FUNCTION_BLOCK LuggageMove (* Basic Function Block Type *)
  (* Standard: 61499-2 *)
  (* Version 0.0, 6/23/2016, Andrei, nxtControl GmbH, Template *)
  PACKAGE Main;
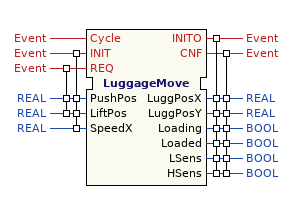
  EVENT_INPUT
    Cycle;
    INIT WITH PushPos, LiftPos, SpeedX; (* Initialization Request *)
    REQ WITH PushPos, LiftPos; (* Normal Execution Request *)
  END_EVENT
  EVENT_OUTPUT
    INITO WITH LuggPosX, LuggPosY, Loading, Loaded, LSens, HSens; (* Initialization Confirm *)
    CNF WITH LuggPosX, LuggPosY, Loading, Loaded, LSens, HSens; (* Execution Confirmation *)
  END_EVENT
  VAR_INPUT
    PushPos : REAL;
    LiftPos : REAL;
    SpeedX : REAL;
  END_VAR
  VAR_OUTPUT
    LuggPosX : REAL; (* Output event qualifier *)
    LuggPosY : REAL;
    Loading : BOOL; (* Input event qualifier *)
    Loaded : BOOL;
    LSens : BOOL;
    HSens : BOOL;
  END_VAR
  VAR
    X : REAL := 0.0;
    Y : REAL := 0.0;
    pPushPos : REAL;
    pLiftPos : REAL;
  END_VAR
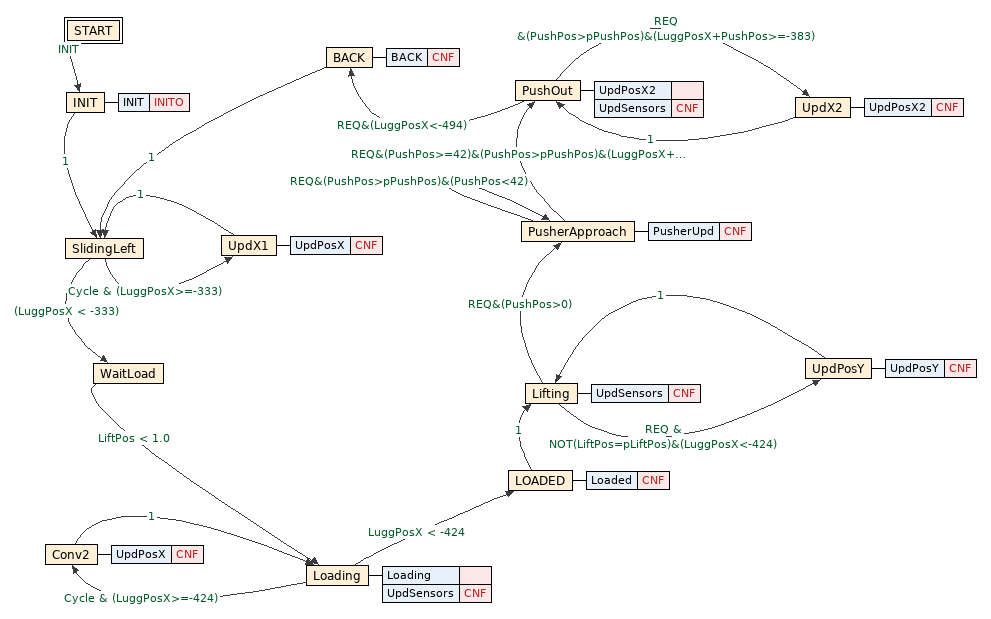
  EC_STATES
    START; (* Initial State *)
    INIT : INIT -> INITO; (* Initialization *)
    SlidingLeft; (* Normal execution *)
    UpdX1 : UpdPosX -> CNF;
    WaitLoad;
    Loading : Loading, UpdSensors -> CNF;
    Conv2 : UpdPosX -> CNF;
    Lifting : UpdSensors -> CNF;
    UpdPosY : UpdPosY -> CNF;
    PushOut : UpdPosX2, UpdSensors -> CNF;
    UpdX2 : UpdPosX2 -> CNF;
    LOADED : Loaded -> CNF;
    PusherApproach : PusherUpd -> CNF;
    BACK : BACK -> CNF;
  END_STATES
  EC_TRANSITIONS
    START TO INIT := INIT;
    INIT TO SlidingLeft := 1;
    SlidingLeft TO UpdX1 := Cycle & (LuggPosX>=-333);
    UpdX1 TO SlidingLeft := 1;
    SlidingLeft TO WaitLoad := (LuggPosX < -333);
    WaitLoad TO Loading := LiftPos < 1.0;
    Loading TO Conv2 := Cycle & (LuggPosX>=-424);
    Conv2 TO Loading := 1;
    Loading TO LOADED := LuggPosX < -424;
    UpdPosY TO Lifting := 1;
    Lifting TO UpdPosY := REQ & NOT(LiftPos=pLiftPos)&(LuggPosX<-424);
    PusherApproach TO PushOut := REQ&(PushPos>=42)&(PushPos>pPushPos)&(LuggPosX+PushPos>=-383);
    PushOut TO UpdX2 := REQ &(PushPos>pPushPos)&(LuggPosX+PushPos>=-383);
    UpdX2 TO PushOut := 1;
    LOADED TO Lifting := 1;
    PusherApproach TO PusherApproach := REQ&(PushPos>pPushPos)&(PushPos<42);
    Lifting TO PusherApproach := REQ&(PushPos>0);
    PushOut TO BACK := REQ&(LuggPosX<-494);
    BACK TO SlidingLeft := 1;
  END_TRANSITIONS
  ALGORITHM INIT IN ST: (* Initialization algorithm *)
X := 0.0;
Y := 0.0;
Loading := FALSE;
Loaded := FALSE;
  END_ALGORITHM
  ALGORITHM UpdPosX IN ST: (* Normally executed algorithm *)
X := X - SpeedX*0.02;
LuggPosX := X;
  END_ALGORITHM
  ALGORITHM Loading IN ST:
Loading := TRUE;
Loaded := FALSE;
  END_ALGORITHM
  ALGORITHM Loaded IN ST:
Loading := FALSE;
Loaded := TRUE;
  END_ALGORITHM
  ALGORITHM UpdPosY IN ST:
LuggPosY := -LiftPos;
pLiftPos:=LiftPos;
  END_ALGORITHM
  ALGORITHM UpdSensors IN ST:
LSens:= (LuggPosY=0) AND (LuggPosX<=-425);
HSens:= (LuggPosY=-150) AND (LuggPosX<=-424) AND (LuggPosX>=-425);
  END_ALGORITHM
  ALGORITHM UpdPosX2 IN ST:
//X := X - SpeedX*0.02;
LuggPosX := -383-PushPos;
pPushPos := PushPos;
  END_ALGORITHM
  ALGORITHM PusherUpd IN ST:
pPushPos := PushPos;
  END_ALGORITHM
  ALGORITHM BACK IN ST:
X := 0.0;
Y := 0.0;
LuggPosX:=0;
LuggPosY:=0;
  END_ALGORITHM
END_FUNCTION_BLOCK
